// TIA Portal V17 export
// export: Created 2025-06-26T07:49:38.6069088Z, ExportSetting WithDefaults, DisplayName Totally Integrated Automation Portal, DisplayVersion V17 Update 8, DisplayName TIA Portal Openness, DisplayVersion V17 Update 8, DisplayName TIA Portal Version Control Interface, DisplayVersion V17, DisplayName STEP 7 Professional, DisplayVersion V17 Update 8, DisplayName STEP 7 Safety, DisplayVersion V17 Update 6, DisplayName WinCC Advanced, DisplayVersion V17 Update 8
FUNCTION_BLOCK "fbFilterDryer"   // FB53, FBD
TITLE = Periodic regulator with a fixed setpoint output
{ S7_Optimized_Access := 'TRUE' }
AUTHOR : Heaten
VERSION : 0.1
// stored: AutoNumber true, IsIECCheckEnabled false, IsRetainMemResEnabled false, MemoryReserve 0, SetENOAutomatically false, UDAEnableTagReadback false
   VAR_INPUT
      bEnable : Bool;
      bReset : Bool;
   END_VAR
   VAR_OUTPUT
      bOut : Bool;
      fOut : Real;
   END_VAR
   VAR_IN_OUT
      sTag : "stFilterDryer";
   END_VAR
   VAR
      Controller : "fbPeriodicRegulator";
   END_VAR
   VAR_TEMP
      bOutput_1 : Bool;
   END_VAR
BEGIN

REGION Network 1: Run regulator
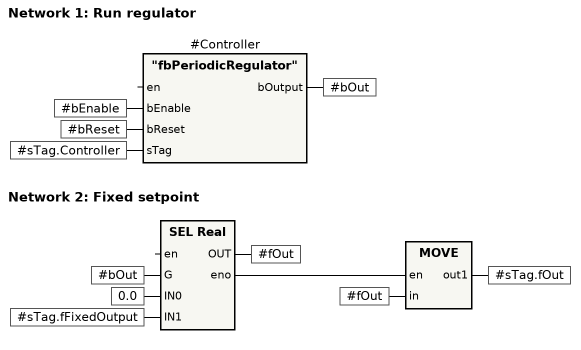
   #Controller(bEnable := #bEnable, bReset := #bReset, sTag := #sTag.Controller, bOutput => #bOut);   // "fbPeriodicRegulator"
END_REGION

REGION Network 2: Fixed setpoint
   // ENO of a box is taken as its EN; it also drops when the box reports an error
   #fOut := SEL(G := #bOut, IN0 := 0.0, IN1 := #sTag.fFixedOutput);
   #sTag.fOut := #fOut;
END_REGION
END_FUNCTION_BLOCK
